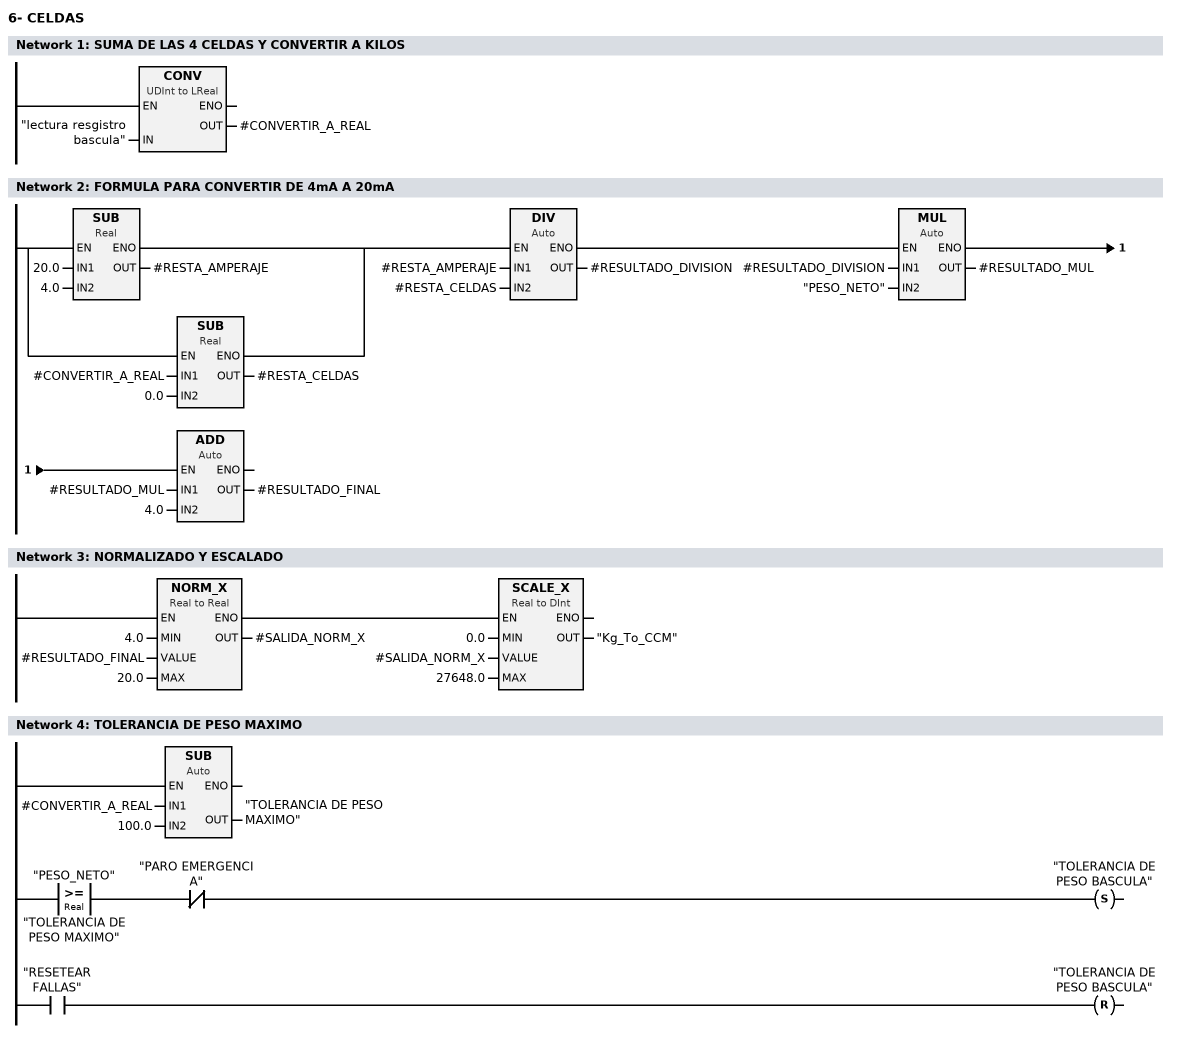
   RUNG wire#powerrail
      { S7_Templates := "[SrcType := UDInt, DestType := LReal]" } Convert(in := "lectura resgistro bascula", out => #CONVERTIR_A_REAL)
   END_RUNG
   // the same network as SCL:
   #CONVERTIR_A_REAL := UDINT_TO_LREAL("lectura resgistro bascula");
END_REGION

REGION Network 2: FORMULA PARA CONVERTIR DE 4mA A 20mA
   RUNG wire#powerrail
      { S7_Templates := "SrcType := Real" } Sub(in1 := 20.0, in2 := 4.0, out => #RESTA_AMPERAJE)
      wire#w1
      Div(in1 := #RESTA_AMPERAJE, in2 := #RESTA_CELDAS, out => #RESULTADO_DIVISION)
      Mul(in1 := #RESULTADO_DIVISION, in2 := "PESO_NETO", out => #RESULTADO_MUL)
      Add(in1 := #RESULTADO_MUL, in2 := 4.0, out => #RESULTADO_FINAL)
   END_RUNG
   RUNG wire#powerrail
      { S7_Templates := "SrcType := Real" } Sub(in1 := #CONVERTIR_A_REAL, in2 := 0.0, out => #RESTA_CELDAS)
   END_RUNG wire#w1
   // the same network as SCL:
   #RESTA_AMPERAJE := 20.0 - 4.0;
   #RESTA_CELDAS := #CONVERTIR_A_REAL - 0.0;
   IF TRUE OR TRUE THEN
       #RESULTADO_DIVISION := #RESTA_AMPERAJE / #RESTA_CELDAS;
       #RESULTADO_MUL := #RESULTADO_DIVISION * "PESO_NETO";
       #RESULTADO_FINAL := #RESULTADO_MUL + 4.0;
   END_IF;
END_REGION

REGION Network 3: NORMALIZADO Y ESCALADO
   RUNG wire#powerrail
      { S7_Templates := "[SrcType := Real, DestType := Real]" } Normalize(min := 4.0, value := #RESULTADO_FINAL, max := 20.0, out => #SALIDA_NORM_X)
      { S7_Templates := "[SrcType := Real, DestType := DInt]" } Scale(min := 0.0, value := #SALIDA_NORM_X, max := 27648.0, out => "Kg_To_CCM")
   END_RUNG
   // the same network as SCL:
   #SALIDA_NORM_X := NORM_X(MIN := 4.0, VALUE := #RESULTADO_FINAL, MAX := 20.0);
   "Kg_To_CCM" := SCALE_X(MIN := 0.0, VALUE := #SALIDA_NORM_X, MAX := 27648.0);
END_REGION

REGION Network 4: TOLERANCIA DE PESO MAXIMO
   RUNG wire#powerrail
      Sub(in1 := #CONVERTIR_A_REAL, in2 := 100.0, out => "TOLERANCIA DE PESO MAXIMO")
   END_RUNG
   RUNG wire#powerrail
      { S7_Templates := "SrcType := Real" } GE_Contact(in1 := "PESO_NETO", in2 := "TOLERANCIA DE PESO MAXIMO")
      I_Contact( "PARO EMERGENCIA" )
      S_Coil( "TOLERANCIA DE PESO BASCULA" )
   END_RUNG
   RUNG wire#powerrail
      Contact( "RESETEAR FALLAS" )
      R_Coil( "TOLERANCIA DE PESO BASCULA" )
   END_RUNG
   // the same network as SCL:
   "TOLERANCIA DE PESO MAXIMO" := #CONVERTIR_A_REAL - 100.0;
   IF ("PESO_NETO" >= "TOLERANCIA DE PESO MAXIMO") AND NOT "PARO EMERGENCIA" THEN
       "TOLERANCIA DE PESO BASCULA" := TRUE;
   END_IF;
   IF "RESETEAR FALLAS" THEN "TOLERANCIA DE PESO BASCULA" := FALSE; END_IF;
END_REGION
END_ORGANIZATION_BLOCK